Yaskawa INFORM job: M-RESET-STATION-2.JBI

/JOB
//NAME M-RESET-STATION-2
//POS
///NPOS 0,0,0,0,0,0
//INST
///DATE 2018/08/23 08:07
///ATTR SC,RW
///GROUP1 ST2
NOP
MRESET ST
END
